// TIA Portal V20 export
DATA_BLOCK "MappingMode_DB"   // DB5
// stored: InstanceOfName Mapping_Mode, InstanceOfType FB
"Mapping_Mode"
   // VAR_INPUT
   //    StateCmd { ExternalAccessible := 'False'; ExternalVisible := 'False'; ExternalWritable := 'False'} : DWord;
   //    ProcedureCur : DWord;
   // END_VAR
   // VAR_OUTPUT
   //    StateFbkIn : DWord;
   // END_VAR
   // VAR
   //    FillingProductionDone : Bool;
   //    DosingProductionDone : Bool;
   //    DosingCleaningDone : Bool;
   // END_VAR
BEGIN
END_DATA_BLOCK
